FUNCTION TryConvert_TIME_TO_ULINT : BOOL
VAR_INPUT
	in : TIME;
	out : REFERENCE TO ULINT;
END_VAR

out := TIME_TO_ULINT(in);
TryConvert_TIME_TO_ULINT := TRUE;

END_FUNCTION

(* stored: Version 1.1.0.1, ProductVersion 3.1.4024.12
   POU TryConvert_TIME_TO_ULINT: Id {44ee1e2d-db85-47ae-8d88-5bb53d741f4b}, SpecialFunc None *)
